// TIA Portal V17 export
// export: Created 2024-09-02T12:49:54.4416756Z, ExportSetting WithDefaults, DisplayName Totally Integrated Automation Portal, DisplayVersion V17, DisplayName TIA Portal Openness, DisplayVersion V17, DisplayName TIA Portal Version Control Interface, DisplayVersion V17, DisplayName STEP 7 Professional, DisplayVersion V17, DisplayName STEP 7 Safety, DisplayVersion V17, DisplayName WinCC Professional, DisplayVersion V17
DATA_BLOCK "AnwDB_F_Diagnose"   // DB7003
TITLE = F-Diagnose
{ S7_Optimized_Access := 'TRUE'; DB_Accessible_From_OPC_UA := 'FALSE' }
AUTHOR : ofuehrus
FAMILY : Safety
NAME : Safety
VERSION : 1.0
// stored: AutoNumber false, DBAccessibleFromOPCUA false, IsOnlyStoredInLoadMemory false, IsRetainMemResEnabled false, IsWriteProtectedInAS false, MemoryReserve 1000
   VAR
      EStop_1 : Byte;   // Not-Halt / emergency stop
      EStop_2 : Byte;   // Not-Halt / emergency stop
      EStop_3 : Byte;   // Not-Halt / emergency stop
      EStop_4 : Byte;   // Not-Halt / emergency stop
      EStop_5 : Byte;   // Not-Halt / emergency stop
      EStop_6 : Byte;   // Not-Halt / emergency stop
      EStop_7 : Byte;   // Not-Halt / emergency stop
      EStop_8 : Byte;   // Not-Halt / emergency stop
      LC_1 : Byte;   // Lichtgitter / light curtain
      LC_2 : Byte;   // Lichtgitter / light curtain
      LC_3 : Byte;   // Lichtgitter / light curtain
      LC_4 : Byte;   // Lichtgitter / light curtain
      LC_5 : Byte;   // Lichtgitter / light curtain
      LC_MUT_1 : Word;   // Lichtgitter mit Muting / Light curtain with muting
      LC_MUT_2 : Word;   // Lichtgitter mit Muting / Light curtain with muting
      LC_MUT_3 : Word;   // Lichtgitter mit Muting / Light curtain with muting
      LC_MUT_4 : Word;   // Lichtgitter mit Muting / Light curtain with muting
      LC_MUT_5 : Word;   // Lichtgitter mit Muting / Light curtain with muting
      SD_1 : Byte;   // Schutzgitter / Safety guard
      SD_2 : Byte;   // Schutzgitter / Safety guard
      SD_3 : Byte;   // Schutzgitter / Safety guard
      SD_4 : Byte;   // Schutzgitter / Safety guard
      SD_5 : Byte;   // Schutzgitter / Safety guard
      BR_1 : Byte;   // Überbrückung / Bridging
      BR_2 : Byte;   // Überbrückung / Bridging
      BR_3 : Byte;   // Überbrückung / Bridging
      BR_4 : Byte;   // Überbrückung / Bridging
      BR_5 : Byte;   // Überbrückung / Bridging
      ReleaseCircuit_01 : Byte;   // Freigabekreis / Relase circuit
      ReleaseCircuit_02 : Byte;   // Freigabekreis / Relase circuit
      ReleaseCircuit_03 : Byte;   // Freigabekreis / Relase circuit
      ReleaseCircuit_04 : Byte;   // Freigabekreis / Relase circuit
      ReleaseCircuit_05 : Byte;   // Freigabekreis / Relase circuit
      ReleaseCircuit_06 : Byte;   // Freigabekreis / Relase circuit
      ReleaseCircuit_07 : Byte;   // Freigabekreis / Relase circuit
      ReleaseCircuit_08 : Byte;   // Freigabekreis / Relase circuit
      ReleaseCircuit_09 : Byte;   // Freigabekreis / Relase circuit
      ReleaseCircuit_10 : Byte;   // Freigabekreis / Relase circuit
      ReleaseCircuit_11 : Byte;   // Freigabekreis / Relase circuit
      ReleaseCircuit_12 : Byte;   // Freigabekreis / Relase circuit
      ReleaseCircuit_13 : Byte;   // Freigabekreis / Relase circuit
      ReleaseCircuit_14 : Byte;   // Freigabekreis / Relase circuit
      ReleaseCircuit_15 : Byte;   // Freigabekreis / Relase circuit
      Protection_Area_1 : Byte;   // Schutzbereich / Scope of protection
      Protection_Area_2 : Byte;   // Schutzbereich / Scope of protection
      Protection_Area_3 : Byte;   // Schutzbereich / Scope of protection
      Protection_Area_4 : Byte;   // Schutzbereich / Scope of protection
      Protection_Area_5 : Byte;   // Schutzbereich / Scope of protection
   END_VAR
BEGIN
END_DATA_BLOCK
